(* IEC 61131-3 sources: StructuredText/, 2 files *)

(* ---- binary_search.st ---- *)
PROGRAM BinarySearch

VAR
target: INT := 10;
list: ARRAY[1..8] OF INT := [1, 2, 5, 10, 12, 15, 17];
left: INT := 1;
right: INT;
result: BOOL;
END_VAR

// Set right to last element in array
right := UPPER_BOUND(list, 1);

result := BinSearch(target, list, left, right)

FUNCTION BinSearch : BOOL
VAR_INPUT
	target : INT;
	list : ARRAY[*] OF INT; //dynamic size array
	left : INT;
	right: INT;
END_VAR

VAR
	midpoint: INT;
END_VAR

// Recusive base case. If left > right target not present
IF left > right THEN
		BinSearch := FALSE;
ELSE
	midpoint := (left + right) / 2;
	// target is midpoint element
	IF list[midpoint] =  target THEN
		BinSearch := TRUE;
	// search left half, target is less than midpoint
	ELSIF target < list[midpoint] THEN
		BinSearch := BinSearch(target, list, left, midpoint - 1);
	// target is greater than midpoint, search right half
	ELSE
		BinSearch(target, list, midpoint + 1, right);
	END_IF

END_FUNCTION

END_PROGRAM

(* ---- prime_number_sieve.st ---- *)
PROGRAM PrimeSieve
VAR
    n: INT := 100; // The upper limit to find primes
    isPrime: ARRAY [1..100] OF BOOL; // Array to hold prime status
    i, j: INT; // Loop counters
END_VAR

// Initialize the array to assume all numbers are prime
FOR i := 1 TO n DO
    isPrime[i] := TRUE;
END_FOR;

// Mark 0 and 1 as not prime
isPrime[1] := FALSE;
isPrime[2] := TRUE;

// Start the sieve algorithm
FOR i := 2 TO n DO
    IF isPrime[i] THEN
        // Mark all multiples of i as not prime
        j := i * 2;
        WHILE j <= n DO
            isPrime[j] := FALSE;
            j := j + i;
        END_WHILE;
    END_IF;
END_FOR;

END_PROGRAM
